ABB RobotStudio station: Solution3_PRUEBA.rsstn

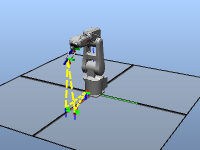
Station Solution3_PRUEBA (saved by RobotStudio 7.0.8504.151)
Controller Controlador1
  mechanical unit ROB_1: IRB120_3_58__01, 6 joints, base frame (0, 0, 0) mm
Layout (positions relative to the parent item):
  - IRB120_3_58__01 [mechanism, from Robots\IRB120_3_58_G_01.rslib] at (0, 0, 0) mm; joint values [0, 0, 0, 0, 0.5236, 0] (rad or m)
  - Mi_mecanismo [mechanism] at (364.35, 0, 594) mm, rotated rx 180 ry 60 rz 180 deg; joint values [0.02, 0.02] (rad or m)
      TCP Mi_mecanismo_1 at (0, -64, -5) mm, rotated rx 0 ry 90 rz -90 deg
      links: bASE, DEDO1, DEDO2
  - Pieza_1 [part] at (488, 79.5, -0.01) mm
Attachment: Mi_mecanismo is attached to IRB120_3_58__01 / Link6
EventTableEntry 1269: Group=, Trigger=DO_pinza 1270, Actions=[EventTableActionMechanicalPose 1271, EventTableActionDetach 1272], Comment=, ActivationMode=2, Cyclic=false
EventTableTriggerIO 1270: IOValue=[0], IRC5Controller=? -1, Operator=0, SignalSource=Controlador1 491
EventTableActionMechanicalPose 1271: VirtualSignal=, Mechanism=Mi_mecanismo 1086, ToPoseName=HomePosition, VirtualSignalValue=[1]
EventTableActionDetach 1272: AttachmentParent=Mi_mecanismo 1086, AttachmentChild=Pieza_1 1108
EventTableTriggerIO 1273: IOValue=[0], IRC5Controller=? -1, Operator=0, SignalSource=Controlador1 491
EventTableTriggerIO 1274: IOValue=[0], IRC5Controller=? -1, Operator=0, SignalSource=Controlador1 491
EventTableTriggerIO 1275: IOValue=[0], IRC5Controller=? -1, Operator=0, SignalSource=Controlador1 491
EventTableTriggerIO 1276: IOValue=[0], IRC5Controller=? -1, Operator=0, SignalSource=Controlador1 491
EventTableTriggerIO 1277: IOValue=[0], IRC5Controller=? -1, Operator=0, SignalSource=Controlador1 491
EventTableTriggerIO 1278: IOValue=[0], IRC5Controller=? -1, Operator=0, SignalSource=Controlador1 491
EventTableTriggerIO 1279: IOValue=[0], IRC5Controller=? -1, Operator=0, SignalSource=Controlador1 491
EventTableEntry 1280: Group=, Trigger=DO_pinza 1281, Actions=[EventTableActionMechanicalPose 1282, EventTableActionAttach 1283], Comment=, ActivationMode=2, Cyclic=false
EventTableTriggerIO 1281: IOValue=[1], IRC5Controller=? -1, Operator=0, SignalSource=Controlador1 491
EventTableActionMechanicalPose 1282: VirtualSignal=, Mechanism=Mi_mecanismo 1086, ToPoseName=POSEFINAL, VirtualSignalValue=[1]
EventTableActionAttach 1283: AttachmentParent=Mi_mecanismo 1086, AttachmentChild=Pieza_1 1108, MountObject=false, Offset=[X=1, Y=0, Z=0, W=0, X=0, Y=1, Z=0, W=0, X=0, Y=0, Z=1, W=0, X=0, Y=0, Z=0, W=1], FlangeIndext=0, FindNearest=false
EventTableTriggerIO 1284: IOValue=[1], IRC5Controller=? -1, Operator=0, SignalSource=Controlador1 491
EventTableTriggerIO 1285: IOValue=[1], IRC5Controller=? -1, Operator=0, SignalSource=Controlador1 491
EventTableTriggerIO 1286: IOValue=[1], IRC5Controller=? -1, Operator=0, SignalSource=Controlador1 491
EventTableTriggerIO 1287: IOValue=[1], IRC5Controller=? -1, Operator=0, SignalSource=Controlador1 491
EventTableTriggerIO 1288: IOValue=[1], IRC5Controller=? -1, Operator=0, SignalSource=Controlador1 491
EventTableTriggerIO 1289: IOValue=[1], IRC5Controller=? -1, Operator=0, SignalSource=Controlador1 491
EventTableTriggerIO 1290: IOValue=[1], IRC5Controller=? -1, Operator=0, SignalSource=Controlador1 491
EventTableTriggerIO 1432: IOValue=[0], IRC5Controller=? -1, Operator=0, SignalSource=Controlador1 491
EventTableTriggerIO 1433: IOValue=[1], IRC5Controller=? -1, Operator=0, SignalSource=Controlador1 491
EventTableTriggerIO 1434: IOValue=[0], IRC5Controller=? -1, Operator=0, SignalSource=Controlador1 491
EventTableTriggerIO 1435: IOValue=[0], IRC5Controller=? -1, Operator=0, SignalSource=Controlador1 491
EventTableTriggerIO 1436: IOValue=[0], IRC5Controller=? -1, Operator=0, SignalSource=Controlador1 491
EventTableTriggerIO 1437: IOValue=[0], IRC5Controller=? -1, Operator=0, SignalSource=Controlador1 491
EventTableTriggerIO 1438: IOValue=[0], IRC5Controller=? -1, Operator=0, SignalSource=Controlador1 491
EventTableTriggerIO 1439: IOValue=[0], IRC5Controller=? -1, Operator=0, SignalSource=Controlador1 491
EventTableTriggerIO 1440: IOValue=[0], IRC5Controller=? -1, Operator=0, SignalSource=Controlador1 491
EventTableTriggerIO 1441: IOValue=[0], IRC5Controller=? -1, Operator=0, SignalSource=Controlador1 491
EventTableTriggerIO 1442: IOValue=[1], IRC5Controller=? -1, Operator=0, SignalSource=Controlador1 491
EventTableTriggerIO 1443: IOValue=[1], IRC5Controller=? -1, Operator=0, SignalSource=Controlador1 491
EventTableTriggerIO 1444: IOValue=[1], IRC5Controller=? -1, Operator=0, SignalSource=Controlador1 491
EventTableTriggerIO 1445: IOValue=[1], IRC5Controller=? -1, Operator=0, SignalSource=Controlador1 491
EventTableTriggerIO 1446: IOValue=[1], IRC5Controller=? -1, Operator=0, SignalSource=Controlador1 491
EventTableTriggerIO 1447: IOValue=[1], IRC5Controller=? -1, Operator=0, SignalSource=Controlador1 491
EventTableTriggerIO 1448: IOValue=[1], IRC5Controller=? -1, Operator=0, SignalSource=Controlador1 491
EventTableTriggerIO 1449: IOValue=[1], IRC5Controller=? -1, Operator=0, SignalSource=Controlador1 491
EventTableTriggerIO 1456: IOValue=[0], IRC5Controller=? -1, Operator=0, SignalSource=Controlador1 491
EventTableTriggerIO 1457: IOValue=[1], IRC5Controller=? -1, Operator=0, SignalSource=Controlador1 491
EventTableTriggerIO 1458: IOValue=[0], IRC5Controller=? -1, Operator=0, SignalSource=Controlador1 491
EventTableTriggerIO 1459: IOValue=[0], IRC5Controller=? -1, Operator=0, SignalSource=Controlador1 491
EventTableTriggerIO 1460: IOValue=[1], IRC5Controller=? -1, Operator=0, SignalSource=Controlador1 491
EventTableTriggerIO 1461: IOValue=[1], IRC5Controller=? -1, Operator=0, SignalSource=Controlador1 491
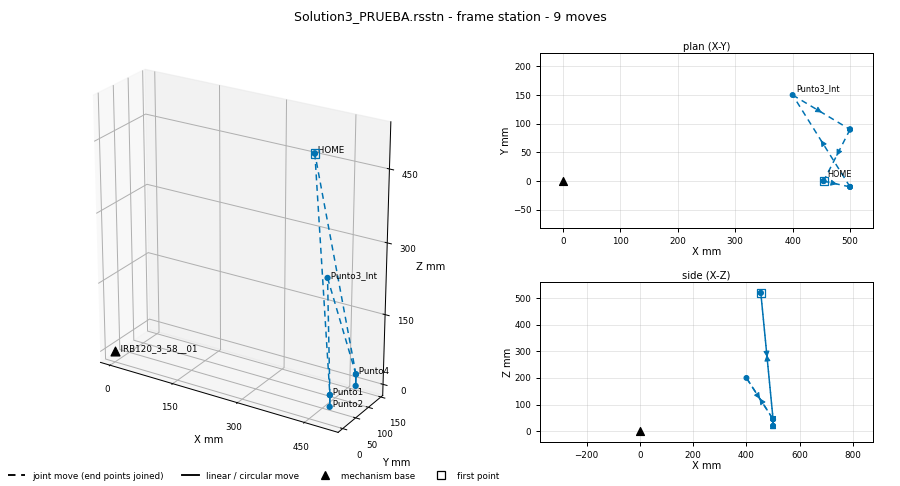
[picture p0: tool path of Solution3_PRUEBA.rsstn in frame station, 9 of 9 moves have a stored position in this frame; points joined in program order, loops and branches not executed]
Targets, tools, work objects and paths stored in the station, written as RAPID:
! task T_ROB1
MODULE CalibData
  TASK PERS wobjdata Workobject_1:=[FALSE,TRUE,"",[[0,0,0],[1,0,0,0]],[[0,0,0],[1,0,0,0]]];
  PERS tooldata Tooldata_1:=[TRUE,[[20,0,115],[1,0,0,0]],[0.5,[1,1,1],[1,0,0,0],0,0,0]];
  PERS tooldata Mi_mecanismo_1:=[TRUE,[[20,0,115],[1,0,0,0]],[0.5,[1,1,1],[1,0,0,0],0,0,0]];
ENDMODULE

! task T_ROB1
MODULE Module1
  CONST robtarget Punto1:=[[500,-10,45],[0,0,1,0],[0,0,0,0],[9E+09,9E+09,9E+09,9E+09,9E+09,9E+09]];
  CONST robtarget Punto2:=[[500,-10,20],[0,0,1,0],[0,0,0,0],[9E+09,9E+09,9E+09,9E+09,9E+09,9E+09]];
  CONST robtarget HOME:=[[453.946750508,0,519.179491924],[0.5,0,0.866025404,0],[0,0,0,0],[9E+09,9E+09,9E+09,9E+09,9E+09,9E+09]];
  CONST robtarget Punto3_Int:=[[400,150,200],[0,0,1,0],[0,0,0,0],[9E+09,9E+09,9E+09,9E+09,9E+09,9E+09]];
  CONST robtarget Punto4:=[[500,90,45],[0,0,1,0],[0,0,0,0],[9E+09,9E+09,9E+09,9E+09,9E+09,9E+09]];
  CONST robtarget Puntofinal:=[[500,90,20],[0,0,1,0],[0,0,0,0],[9E+09,9E+09,9E+09,9E+09,9E+09,9E+09]];
  PROC Path_10()
    MoveJ HOME,v200,fine,Mi_mecanismo_1\WObj:=Workobject_1;
    Reset DO_pinza;
    MoveJ Punto1,v200,fine,Mi_mecanismo_1\WObj:=Workobject_1;
    MoveL Punto2,v100,fine,Mi_mecanismo_1\WObj:=Workobject_1;
    Set DO_pinza;
    MoveL Punto1,v100,fine,Mi_mecanismo_1\WObj:=Workobject_1;
    MoveJ Punto3_Int,v200,fine,Mi_mecanismo_1\WObj:=Workobject_1;
    MoveJ Punto4,v200,fine,Mi_mecanismo_1\WObj:=Workobject_1;
    MoveL Puntofinal,v100,fine,Mi_mecanismo_1\WObj:=Workobject_1;
    Reset DO_pinza;
    MoveL Punto4,v100,fine,Mi_mecanismo_1\WObj:=Workobject_1;
    MoveJ HOME,v400,fine,Mi_mecanismo_1\WObj:=Workobject_1;
  ENDPROC
ENDMODULE

